// TIA Portal V17 export
// export: Created 2025-03-05T08:02:53.1431431Z, ExportSetting WithDefaults, DisplayName Totally Integrated Automation Portal, DisplayVersion V17 Update 8, DisplayName TIA Portal Openness, DisplayVersion V17 Update 8, DisplayName TIA Portal Version Control Interface, DisplayVersion V17, DisplayName SINAMICS Startdrive Advanced, DisplayVersion V17 SP2, DisplayName SINAMICS Startdrive G110M, G120, G120C, G120D, G120P, G115D, DisplayVersion V17 SP2, DisplayName SINAMICS Startdrive G130, G150, S120, S150, SINAMICS MV, S210, DisplayVersion V17 SP2, DisplayName STEP 7 Professional, DisplayVersion V17 Update 8, DisplayName SINUMERIK ONE STEP 7 Toolbox, DisplayVersion V17 Update 12, DisplayName SINUMERIK 840D sl STEP 7 Toolbox, DisplayVersion V17 Update 12, DisplayName STEP 7 Safety, DisplayVersion V17 Update 6, DisplayName WinCC Advanced, DisplayVersion V17 Update 8
DATA_BLOCK "DB7800_HMI_HOPPER_ACTIONS"   // DB7800
{ S7_Optimized_Access := 'TRUE'; DB_Accessible_From_OPC_UA := 'FALSE' }
VERSION : 0.1
// stored: AutoNumber false, DBAccessibleFromOPCUA false, DBAccessibleFromWebserver true, IsOnlyStoredInLoadMemory false, IsRetainMemResEnabled false, IsWriteProtectedInAS false, MemoryReserve 0
   VAR
      ARRAY_STIRRER_SPEED_MANUAL_START : Array[0..4] of Bool;
      ARRAY_FEEDING_COVER_MANUAL_START : Array[0..4] of Bool;
      ARRAY_HOPPER_COVER_MANUAL_START : Array[0..4] of Bool;
      ARRAY_UPPER_JACKET_MANUAL_START : Array[0..4] of Bool;
      ARRAY_LOWER_JACKET_MANUAL_START : Array[0..4] of Bool;
      ARRAY_STIRRER_SPEED_MANUAL_STOP : Array[0..4] of Bool;
      ARRAY_FEEDING_COVER_MANUAL_STOP : Array[0..4] of Bool;
      ARRAY_HOPPER_COVER_MANUAL_STOP : Array[0..4] of Bool;
      ARRAY_UPPER_JACKET_MANUAL_STOP : Array[0..4] of Bool;
      ARRAY_LOWER_JACKET_MANUAL_STOP : Array[0..4] of Bool;
   END_VAR
BEGIN
END_DATA_BLOCK
